PROGRAM Carriage_Manager
VAR
	Carriage_Offset: LREAL; //general offset of the encoder value
	VeloManJog: REAL := 5; //speed of the regular jog movement
	VeloManJogFAST: REAL := 60; // speed of the fast movement
	
	ExtraSensorInput: TAxSensorModule; // compressed FUN for exteriour sensor inputs. temp, edge, jog stops
	SpecialOperations: TAxSpecialOperationModule; //compressed FUN for the special operation commands. 
	AxisCoupleIN: TAxCoupleModule; //connects to the AX_Couple_out of the manager from the next axis. NOT MASTER/SLAVE
	ErrorWordArray: WORD; //build a array of words that act as a cluster of error watching variables. each step in array will be one axis. differant values of the word for each axis mean a differant error. 
	JogStop: LREAL := 1E100 ; // a stopping point using the jog system to signify it is in the right spot. Need to have the LimitPosJOG adjusted after to compensate for the next space.
	DriveCMD_1: DriveCMDShortCUT; //extra system for the FB to make it easy to read.
	ASPshortCut_1: ASPshortCUT;  // same as above
END_VAR

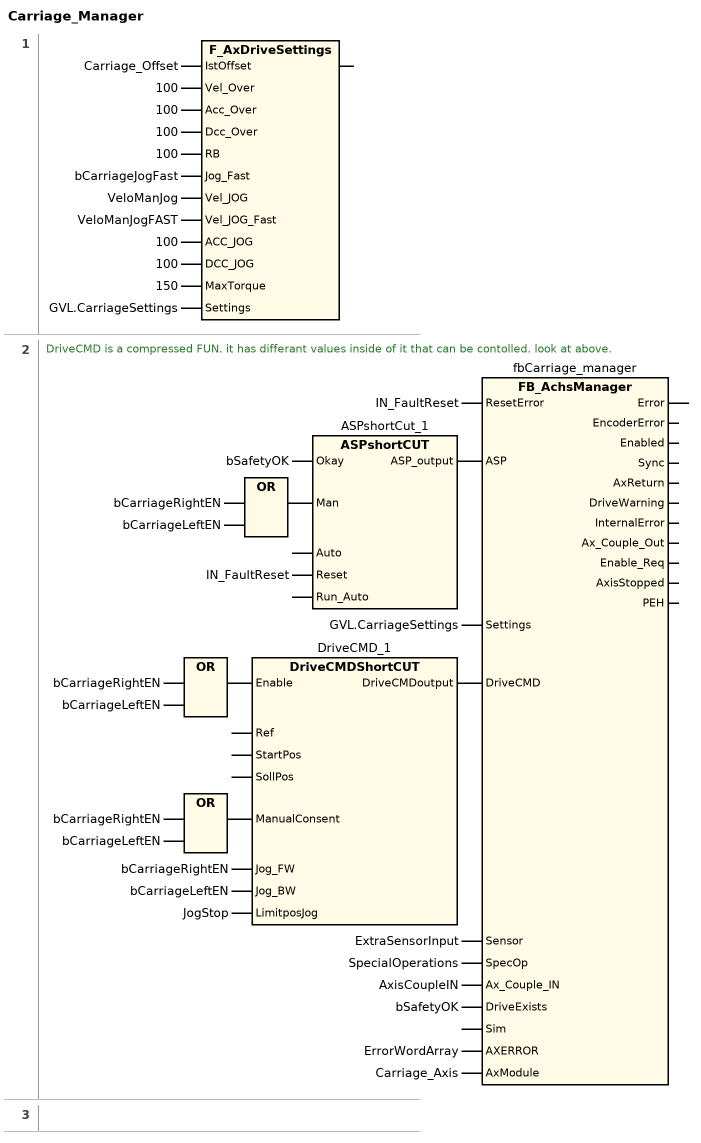
// NETWORK 1
F_AxDriveSettings(IstOffset := Carriage_Offset, Vel_Over := 100, Acc_Over := 100, Dcc_Over := 100, RB := 100, Jog_Fast := bCarriageJogFast, Vel_JOG := VeloManJog, Vel_JOG_Fast := VeloManJogFAST, ACC_JOG := 100, DCC_JOG := 100, MaxTorque := 150, Settings := GVL.CarriageSettings);

// NETWORK 2
// DriveCMD is a compressed FUN. it has differant values inside of it that can be contolled. look at above.
ASPshortCut_1(Okay := bSafetyOK, Man := bCarriageRightEN OR bCarriageLeftEN, Reset := IN_FaultReset); // ASPshortCUT
DriveCMD_1(
    Enable := bCarriageRightEN OR bCarriageLeftEN,
    ManualConsent := bCarriageRightEN OR bCarriageLeftEN,
    Jog_FW := bCarriageRightEN,
    Jog_BW := bCarriageLeftEN,
    LimitposJog := JogStop); // DriveCMDShortCUT
fbCarriage_manager(
    ResetError := IN_FaultReset,
    ASP := ASPshortCut_1.ASP_output,
    Settings := GVL.CarriageSettings,
    DriveCMD := DriveCMD_1.DriveCMDoutput,
    Sensor := ExtraSensorInput,
    SpecOp := SpecialOperations,
    Ax_Couple_IN := AxisCoupleIN,
    DriveExists := bSafetyOK,
    AXERROR := ErrorWordArray,
    AxModule := Carriage_Axis); // FB_AchsManager

// NETWORK 3

END_PROGRAM

(* stored: Version 1.1.0.1, ProductVersion 3.1.4024.15
   POU Carriage_Manager: Id {39878625-31a5-4a62-950b-d6dbf2d5e968}, SpecialFunc None *)
